FUNCTION_BLOCK BargraphSplitFS_AR (* AR adapter wrapper around BargraphSplitFS — accepts the signed value via AR adapter socket instead of a plain REQ/rValue pair *)
  (* Standard: ISO 11783-6; Description: Copyright (c) 2026 Meisterschulen am Ostbahnhof This program and the accompanying materials are made available under the terms of the Eclipse Public License 2.0 which is available at https://www.eclipse.org/legal/epl-2.0/ SPDX-License-Identifier: EPL-2.0 Same wrapper shape as PositionMarkerFSA around PositionMarkerFS: the AR adapter socket's value drives the internally-owned BargraphSplitFS instance's REQ/rValue directly. xOverRight/xOverLeft are re-exposed as AX adapter plugs, exactly like PositionMarkerFSA does for xOver/xUnder. *)
  (* Version 1.0, 2026-09-05, Franz Höpfinger, Meisterschulen am Ostbahnhof, initial API and implementation and/or initial documentation *)
  PACKAGE isobus::UT::Q;
  IMPORT isobus::utils::bargraph::BargraphSplit_S;
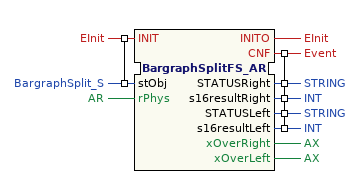
  EVENT_INPUT
    INIT : EInit WITH stObj; (* Service Initialization *)
  END_EVENT
  EVENT_OUTPUT
    INITO : EInit; (* Initialization Confirm *)
    CNF WITH STATUSRight, s16resultRight, STATUSLeft, s16resultLeft; (* Confirmation of Requested Service *)
  END_EVENT
  VAR_INPUT
    stObj : isobus::utils::bargraph::BargraphSplit_S; (* Split-bargraph object pool properties (left/right Bargraph refs, shared magnitude bounds), snapshotted at INIT *)
  END_VAR
  VAR_OUTPUT
    STATUSRight : STRING; (* Service Status - passthrough from the internal BargraphSplitFS *)
    s16resultRight : INT; (* retval - passthrough from the internal BargraphSplitFS *)
    STATUSLeft : STRING; (* Service Status - passthrough from the internal BargraphSplitFS *)
    s16resultLeft : INT; (* retval - passthrough from the internal BargraphSplitFS *)
  END_VAR
  SOCKETS
    rPhys : adapter::types::unidirectional::AR; (* Signed physical value input *)
  END_SOCKETS
  PLUGS
    xOverRight : adapter::types::unidirectional::AX; (* rValue exceeded stObj.r32MaxMagnitude and the right side was clamped *)
    xOverLeft : adapter::types::unidirectional::AX; (* -rValue exceeded stObj.r32MaxMagnitude and the left side was clamped *)
  END_PLUGS
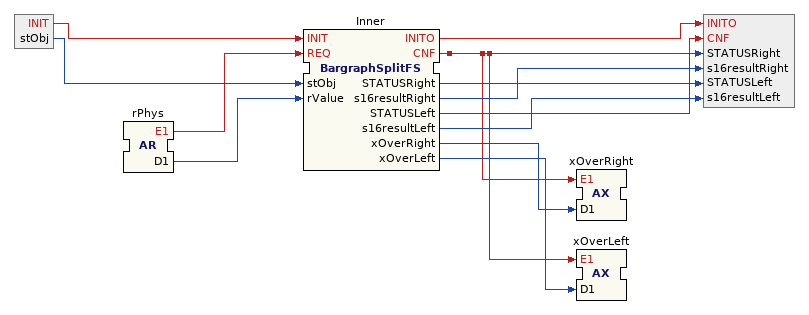
  FBS
    Inner : isobus::UT::Q::BargraphSplitFS;
  END_FBS
  EVENT_CONNECTIONS
    INIT TO Inner.INIT;
    rPhys.E1 TO Inner.REQ;
    Inner.INITO TO INITO;
    Inner.CNF TO CNF;
    Inner.CNF TO xOverRight.E1;
    Inner.CNF TO xOverLeft.E1;
  END_CONNECTIONS
  DATA_CONNECTIONS
    stObj TO Inner.stObj;
    rPhys.D1 TO Inner.rValue;
    Inner.STATUSRight TO STATUSRight;
    Inner.s16resultRight TO s16resultRight;
    Inner.STATUSLeft TO STATUSLeft;
    Inner.s16resultLeft TO s16resultLeft;
    Inner.xOverRight TO xOverRight.D1;
    Inner.xOverLeft TO xOverLeft.D1;
  END_CONNECTIONS
END_FUNCTION_BLOCK
